# EPICS autosave request: iocBoot/iocTomoScan_2BM/auto_settings.req
file "tomoScan_settings.req", P=$(P), R=$(R)
file "tomoScan_PSO_settings.req", P=$(P), R=$(R)
file "tomoScan_2BM_settings.req", P=$(P), R=$(R)
